FUNCTION F_DecimalData : LREAL
VAR_INPUT
	
	//
	data_type : STRING;
	//
	value_input : LREAL;
	
	// decimal places
	n_decimal_digit : INT;
	
	// Round or not
	b_round: BOOL;
	
	// variable for comparison 
	//n_temp_INT : ANY_INT;
	//f_temp_REAL : ANY_REAL;
	//f_temp_LREAL : ANY_REAL;
END_VAR
	
VAR
	value_Output : LREAL;

END_VAR


// This Function is for decimal the data by data type
// only for OUTPUT LREAL and now 

IF data_type = 'REAL' THEN
	
	value_Output:= STRING_TO_REAL(LREAL_TO_FMTSTR(TO_LREAL(value_input), n_decimal_digit, b_round));
	
ELSIF data_type = 'LREAL' THEN
	
	value_Output:= STRING_TO_REAL(LREAL_TO_FMTSTR(value_input, n_decimal_digit, b_round));
	
END_IF

END_FUNCTION

(* stored: Version 1.1.0.1, ProductVersion 3.1.4024.11
   POU F_DecimalData: Id {66d33ad8-e83a-4919-8f59-cd46dd00ddc3}, SpecialFunc None *)
